TYPE st_language :
STRUCT
	portuguese				:BOOL:=FALSE;
	english					:BOOL:=TRUE;
END_STRUCT
END_TYPE

(* stored: Version 1.1.0.1, ProductVersion 3.1.4020.12
   DUT st_language: Id {4d14fcd5-f410-4e5e-bcbf-84743af48247} *)
